Staubli VAL3: SETFRAME.pgx

public program SetFrame(trsf& x_trSource[], frame& x_fFrame, bool& x_bRes)
  local point l_pPoint[3]
  local num l_ni
  local bool l_bIn
begin
  //把三个trsf转换为frame
  //如果x_frame是局部变量,需要在建立的程序中先link
  link(x_fFrame,world)
  x_fFrame.trsf={0,0,0,0,0,0}
  x_bRes=false
  if size(x_trSource)<3
    return
  endIf


  //建立frame
  for l_ni=0 to 2
    l_pPoint[l_ni].trsf=x_trSource[l_ni]
    link(l_pPoint[l_ni],world)
  endFor

  x_bRes=setFrame(l_pPoint[0],l_pPoint[1],l_pPoint[2],x_fFrame)==0


end
